FUNCTION AlarmCheck : BOOL
VAR_INPUT
	AlarmSet : BOOL; (*Check if alarm is set*)
END_VAR

IF AlarmSet THEN
	AlarmCheck := TRUE; // Alarm goes off
ELSE
	AlarmCheck := FALSE; // Alarm doesn't go off	
END_IF

END_FUNCTION

(* stored: Version 1.1.0.1, ProductVersion 3.1.4024.12
   POU AlarmCheck: Id {6a364238-c05e-42c3-a3fc-b9d78f1103e6}, SpecialFunc None *)
